(* PLC project Evolved Test, FAszom KFT TEST PLC Program 0.1.23.456 *)
(* stored: creationDateTime 1990-01-01T12:00:00, modificationDateTime 2016-04-10T17:37:00 *)

PROGRAM MotorExample
  VAR
    state : INT := 1;
    Distance : LREAL := 360;
    PowerX : MC_Power;
    Xonb : BOOL;
    HomeX : MC_Home;
    Referenced : BOOL;
    ExtendX : MC_MoveRelative;
    Wait : TON;
    RetractX : MC_MoveAbsolute;
    Wait_time : TIME := TIME#3s0ms;
    Elapsed_time : TIME;
    ResetX : MC_Reset;
    ReadAxisState : MC_ReadStatus;
    Xerrorstop : BOOL;
    XerrorID : DWORD;
    Counter : INT := 0;
  END_VAR
  VAR CONSTANT
    ERROR : INT := 99;
  END_VAR

                    
CASE state OF
	
1:
PowerX(
	Axis:=MotorExample_Motor , 
	Enable:=TRUE , 
	bRegulatorOn:=TRUE , 
	bDriveStart:=TRUE , 
	Status=> , 
	bRegulatorRealState=> , 
	bDriveStartRealState=> , 
	Busy=> , 
	Error=> , 
	ErrorID=> );
	
	IF PowerX.bDriveStartRealState THEN
		Xonb:=TRUE;
		state:=state+1;
		ELSE
			state:=ERROR;
	END_IF
	
2:
HomeX(
	Axis:=MotorExample_Motor , 
	Execute:=TRUE, 
	Position:=0.0, 
	Done=> , 
	Busy=> , 
	CommandAborted=> , 
	Error=> , 
	ErrorID=> );
		
	IF HomeX.Done THEN
		Referenced:=TRUE;
		state:=state+1;
		HomeX.Execute:=FALSE;
		ELSIF HomeX.Error OR Xerrorstop OR MotorExample_Motor.bError THEN
		state:=ERROR;
	END_IF
	
3:
ExtendX.Execute:=TRUE; 
ExtendX.Distance:=Distance; 
ExtendX.Velocity:=100; 
ExtendX.Acceleration:=1000; 
ExtendX.Deceleration:=1000; 
ExtendX.Jerk:=0; 

	IF ExtendX.Done THEN
		state:=state+1;
		ExtendX.Execute:=FALSE;
		ELSIF ExtendX.Error OR Xerrorstop OR MotorExample_Motor.bError THEN
		state:=ERROR;	
	END_IF
	
4:
Wait.IN:=TRUE;
Wait.PT:=Wait_time;
Elapsed_time:=Wait.ET;

	IF Wait.Q THEN
		state:=state+1;
		Wait.IN:=FALSE;
	END_IF

5: 
RetractX.Execute:=TRUE; 
RetractX.Position:=0; 
RetractX.Velocity:=100;
RetractX.Acceleration:=1000;
RetractX.Deceleration:=1000; 
RetractX.Jerk:=0; 

IF RetractX.Done THEN
		state:=state+1;
		RetractX.Execute:=FALSE;
		counter:=counter+1;
		ELSIF RetractX.Error OR Xerrorstop THEN
		state:=ERROR;
	END_IF
	
6: 
Wait.IN:=TRUE; 
Wait.PT:=Wait_time;
Elapsed_time:=Wait.ET;

	IF Wait.Q THEN
		state:=3;
		Wait.IN:=FALSE;
	END_IF
	
ERROR:
ResetX.Execute:=TRUE;
Wait.IN:=TRUE;
IF Wait.Q THEN
	ResetX.Execute:=FALSE;
	state:=1;
END_IF

END_CASE
ExtendX(Axis:=MotorExample_Motor);
Wait();
RetractX(Axis:=MotorExample_Motor);
ResetX(Axis:=MotorExample_Motor);
ReadAxisState(Axis:=MotorExample_Motor,Enable:=TRUE,ErrorStop=>Xerrorstop);




                  
END_PROGRAM

PROGRAM Motor_Proba
  VAR_INPUT
    START AT %MX0.1 : BOOL := FALSE;
    STOP AT %MX0.2 : BOOL := FALSE;
  END_VAR
  VAR
    MOTOR AT %MX1.0 : BOOL := FALSE;
    ERROR AT %MX2.0 : BOOL := FALSE;
  END_VAR
  VAR
    ERR_TIM : TON;
    EL_TIME : TIME;
  END_VAR
  VAR_OUTPUT
    ST_RED AT %QX1.1 : BOOL;
    ST_GREEN AT %QX3.1 : BOOL;
  END_VAR

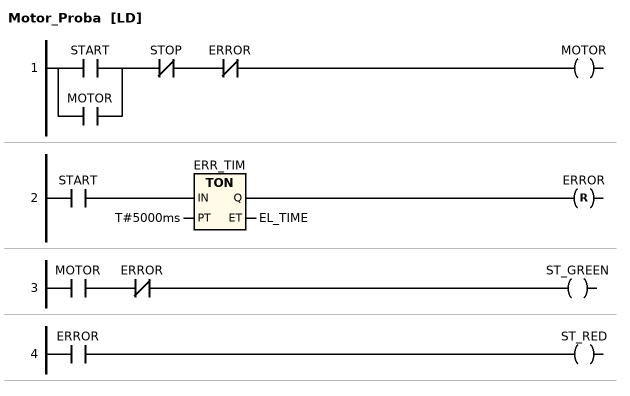
(* LD diagram, written out as Structured Text *)

MOTOR := (START OR MOTOR) AND NOT STOP AND NOT ERROR;

ERR_TIM(IN := START, PT := T#5000ms, ET => EL_TIME);
IF ERR_TIM.Q THEN ERROR := FALSE; END_IF;

ST_GREEN := MOTOR AND NOT ERROR;

ST_RED := ERROR;
END_PROGRAM

PROGRAM St_xample
  VAR
    input AT %MX3.3 : BOOL;
    output AT %QX0.1 : BOOL;
  END_VAR

									
									output := input;
									
								
END_PROGRAM

(* @NESTEDCOMMENTS := 'Yes' @PATH := '' @SYMFILEFLAGS := '2048' *)
FUNCTION_BLOCK fuzzy_exp
  VAR_INPUT
    PV : REAL;
    SP : REAL;
    MV_LN : REAL;
    MV_MN : REAL;
    MV_SN : REAL;
    MV_SP : REAL;
    MV_MP : REAL;
    MV_LP : REAL;
    LN_Error_Rate : REAL;
    MN_Error_Rate : REAL;
    MP_Error_Rate : REAL;
    LP_Error_Rate : REAL;
    Update_Time : WORD;
    Manual : BOOL;
    CV_Manual : REAL;
    CV_Min : REAL;
    CV_Max : REAL;
    Enable : BOOL;
  END_VAR
  VAR_OUTPUT
    FL_CV : REAL;
  END_VAR
  VAR
    Loop_Update_ONS : R_TRIG;
    Loop_Update_Trigger : BOOL;
    TMR_Loop_Update : TON;
    Loop_Update_Time : WORD;
    Loop_Update_mSec : TIME;
    Process_Error : REAL;
    NL_Error : BOOL;
    NM_Error : BOOL;
    NS_Error : BOOL;
    PS_Error : BOOL;
    PM_Error : BOOL;
    PL_Error : BOOL;
    Process_Error_Rate : REAL;
    Error_Rate_PV1 : REAL;
    Error_Rate_PV2 : REAL;
    NL_Error_Rate_Ind : BOOL;
    NM_Error_Rate_Ind : BOOL;
    NS_Error_Rate_Ind : BOOL;
    PS_Error_Rate_Ind : BOOL;
    PM_Error_Rate_Ind : BOOL;
    PL_Error_Rate_Ind : BOOL;
    Output_CV : REAL;
  END_VAR

                    (* @END_DECLARATION := '0' *)
(****************************************************************************************************************************
	POU Title:  	Fuzzy_Logic(PRG)
   
 	Designer:	K. Presssley
	Date:		01/09/09
		
	Function:	The function of this program is to implement a fuzzy logic control algorithm for process control..  
****************************************************************************************************************************)
(***** Loop Update Logic *****)
(*  Get the Loop Update Time, ensure that lower limit of 1 is not exceeded and convert it into a time variable  *)
	IF Update_Time < 1 THEN
		Loop_Update_Time := 1;
	ELSE
		Loop_Update_Time := Update_Time;
	END_IF;

	Loop_Update_mSec := WORD_TO_TIME(Loop_Update_Time);

	IF NOT TMR_Loop_Update.Q THEN
		Loop_Update_Trigger := TRUE;
	ELSE
		Loop_Update_Trigger := FALSE;
	END_IF;

	TMR_Loop_Update( IN := Loop_Update_Trigger, PT:= Loop_Update_mSec );
 	  Loop_Update_ONS( CLK := TMR_Loop_Update.Q);



(***** Calculate the Process Error and Process Error Rate *****)
	IF Loop_Update_ONS.Q THEN
	  (* Process Error Calculation *)
		Process_Error := SP - PV;

	  (* Process Error Rate Calculation *)
	 	Error_Rate_PV1 := Error_Rate_PV2;
		  Error_Rate_PV2 := PV;
		   Process_Error_Rate := (Error_Rate_PV2 - Error_Rate_PV1) / (Loop_Update_Time);
	END_IF;


(***** Membership Zone Logic *****)
(* Error Zone Identification Logic - This logic will indentify which Error Zone the Process Value is currently in *)
	(* Negative Large Membership Zone *)
		IF Process_Error <= MV_LN THEN
			NL_Error := TRUE;
		ELSE
			NL_Error := FALSE;
		END_IF;

	(* Negative Medium Membership Zone *)
		IF Process_Error > MV_LN AND Process_Error <= MV_MN THEN
			NM_Error := TRUE;
		ELSE
			NM_Error := FALSE;
		END_IF;

	(* Negative Small Membership Zone *)
		IF Process_Error > MV_MN AND Process_Error <= MV_SN THEN
			NS_Error := TRUE;
		ELSE
			NS_Error := FALSE;
		END_IF;

	(* Positive Small Membership Zone *)
		IF Process_Error < MV_MP AND Process_Error >= MV_SP THEN
			PS_Error := TRUE;
		ELSE
			PS_Error := FALSE;
		END_IF;

	(* Positive Medium Membership Zone *)
		IF Process_Error < MV_LP AND Process_Error >= MV_MP THEN
			PM_Error := TRUE;
		ELSE
			PM_Error := FALSE;
		END_IF;

	(* Positive Large Membership Zone *)
		IF Process_Error >= MV_LP THEN
			PL_Error := TRUE;
		ELSE
			PL_Error := FALSE;
		END_IF;

(* Error Rate Zone Identification Logic - This logic will indentify which Error Rate Zone the Process Value is currently in *)
	(* Negative Large Error Rate Membership Zone - The Error Rate is Decreasing Quickly *)
		IF Process_Error_Rate <= LN_Error_Rate THEN
			NL_Error_Rate_Ind := TRUE;
		ELSE
			NL_Error_Rate_Ind := FALSE;
		END_IF;

	(* Negative Medium Error Rate Membership Zone - The Error Rate is Decreasing *)
		IF Process_Error_Rate > LN_Error_Rate AND Process_Error_Rate <= MN_Error_Rate THEN
			NM_Error_Rate_Ind := TRUE;
		ELSE
			NM_Error_Rate_Ind := FALSE;
		END_IF;

	(* Negative Small Error Rate Membership Zone  - The Error Rate is Decreasing slowly *)
		IF Process_Error_Rate > MN_Error_Rate AND Process_Error_Rate < 0.0 THEN
			NS_Error_Rate_Ind := TRUE;
		ELSE
			NS_Error_Rate_Ind := FALSE;
		END_IF;

	(* Positive Small Error Rate Membership Zone  - The Error Rate is Increasing slowly *)
		IF Process_Error_Rate < MP_Error_Rate AND Process_Error_Rate >= 0.0 THEN
			PS_Error_Rate_Ind := TRUE;
		ELSE
			PS_Error_Rate_Ind := FALSE;
		END_IF;

	(* Positive Meduim Error Rate Membership Zone  - The Error Rate is Increasing *)
		IF Process_Error_Rate < LP_Error_Rate AND Process_Error_Rate >= MP_Error_Rate THEN
			PM_Error_Rate_Ind := TRUE;
		ELSE
			PM_Error_Rate_Ind := FALSE;
		END_IF;

	(* Positive Large Error Rate Membership Zone  - The Error Rate is Increasing Quickly  *)
		IF Process_Error_Rate >= LP_Error_Rate THEN
			PL_Error_Rate_Ind := TRUE;
		ELSE
			PL_Error_Rate_Ind := FALSE;
		END_IF;


(***** Fuzzy Logic Rules *****)
(* This section of logic contains all of the Fuzzy Logic rules required to produce the control action *)
	(* PV is Far Above SP and Increasing Quickly *)
		IF Loop_Update_ONS.Q AND NL_Error AND PL_Error_Rate_Ind
		    AND Enable AND NOT Manual THEN
			Output_CV := Output_CV - 1000.0;
		END_IF;

	(* PV is Far Above SP and Increasing *)
		IF Loop_Update_ONS.Q AND NL_Error AND PM_Error_Rate_Ind
		    AND Enable AND NOT Manual THEN
			Output_CV := Output_CV - 300.0;
		END_IF;

	(* PV is Far Above SP and Increasing slowly *)
		IF Loop_Update_ONS.Q AND NL_Error AND PS_Error_Rate_Ind
		    AND Enable AND NOT Manual THEN
			Output_CV := Output_CV - 250.0;
		END_IF;

	(* PV is Far Above SP and Decreasing slowly *)
		IF Loop_Update_ONS.Q AND NL_Error AND NS_Error_Rate_Ind
		    AND Enable AND NOT Manual THEN
			Output_CV := Output_CV - 300;
		END_IF;

	(* PV is Far Above SP and Decreasing *)
		IF Loop_Update_ONS.Q AND NL_Error AND NM_Error_Rate_Ind
		    AND Enable AND NOT Manual THEN
			Output_CV := Output_CV - 250.0;
		END_IF;

	(* PV is Far Above SP and Decreasing Quickly *)
		IF Loop_Update_ONS.Q AND NL_Error AND NL_Error_Rate_Ind
		    AND Enable AND NOT Manual THEN
			Output_CV := Output_CV - 100.0;
		END_IF;

	(* PV is Above SP and Increasing Quickly *)
		IF Loop_Update_ONS.Q AND NM_Error AND PL_Error_Rate_Ind
		    AND Enable AND NOT Manual THEN
			Output_CV := Output_CV - 250.0;
		END_IF;

	(* PV is Above SP and Increasing *)
		IF Loop_Update_ONS.Q AND NM_Error AND PM_Error_Rate_Ind
		    AND Enable AND NOT Manual THEN
			Output_CV := Output_CV - 100.0;
		END_IF;

	(* PV is Above SP and Increasing slowly *)
		IF Loop_Update_ONS.Q AND NM_Error AND PS_Error_Rate_Ind
		    AND Enable AND NOT Manual THEN
			Output_CV := Output_CV - 50.0;
		END_IF;

	(* PV is Above SP and Decreasing Slowly *)
		IF Loop_Update_ONS.Q AND NM_Error AND NS_Error_Rate_Ind
		    AND Enable AND NOT Manual THEN
			Output_CV := Output_CV - 250.0;
		END_IF;

	(* PV is Above SP and Decreasing *)
		IF Loop_Update_ONS.Q AND NM_Error AND NM_Error_Rate_Ind
		    AND Enable AND NOT Manual THEN
			Output_CV := Output_CV - 100.0;
		END_IF;

	(* PV is Above SP and Decreasing Quickly *)
		IF Loop_Update_ONS.Q AND NM_Error AND NL_Error_Rate_Ind
		    AND Enable AND NOT Manual THEN
			Output_CV := Output_CV - 50.0;
		END_IF;

	(* PV is Slightly Above SP and Increasing Quickly *)
		IF Loop_Update_ONS.Q AND NS_Error AND PL_Error_Rate_Ind
		    AND Enable AND NOT Manual THEN
			Output_CV := Output_CV - 20.0;
		END_IF;

	(* PV is Slightly Above SP and Increasing *)
		IF Loop_Update_ONS.Q AND NS_Error AND PM_Error_Rate_Ind
		    AND Enable AND NOT Manual THEN
			Output_CV := Output_CV - 10.0;
		END_IF;

	(* PV is Slightly Above SP and Increasing slowly*)
		IF Loop_Update_ONS.Q AND NS_Error AND PS_Error_Rate_Ind
		    AND Enable AND NOT Manual THEN
			Output_CV := Output_CV - 5.0;
		END_IF;

	(* PV is Slightly Above SP and Decreasing slowly*)
		IF Loop_Update_ONS.Q AND NS_Error AND NS_Error_Rate_Ind
		    AND Enable AND NOT Manual THEN
			Output_CV := Output_CV - 20.0;
		END_IF;

	(* PV is Slightly Above SP and Decreasing *)
		IF Loop_Update_ONS.Q AND NS_Error AND NM_Error_Rate_Ind
		    AND Enable AND NOT Manual THEN
			Output_CV := Output_CV - 10.0;
		END_IF;

	(* PV is Slightly Above SP and Decreasing Quickly*)
		IF Loop_Update_ONS.Q AND NS_Error AND NL_Error_Rate_Ind
		    AND Enable AND NOT Manual THEN
			Output_CV := Output_CV - 5.0;
		END_IF;

	(* PV is Slightly Below SP and Increasing Quickly *)
		IF Loop_Update_ONS.Q AND PS_Error AND PL_Error_Rate_Ind
		    AND Enable AND NOT Manual THEN
			Output_CV := Output_CV + 5.0;
		END_IF;

	(* PV is Slightly Below SP and Increasing *)
		IF Loop_Update_ONS.Q AND PS_Error AND PM_Error_Rate_Ind
		    AND Enable AND NOT Manual THEN
			Output_CV := Output_CV + 10.0;
		END_IF;

	(* PV is Slightly Below SP and Increasing Slowly *)
		IF Loop_Update_ONS.Q AND PS_Error AND PS_Error_Rate_Ind
		    AND Enable AND NOT Manual THEN
			Output_CV := Output_CV + 20.0;
		END_IF;

	(* PV is Slightly Below SP and Decreasing Slowly *)
		IF Loop_Update_ONS.Q AND PS_Error AND NS_Error_Rate_Ind
		    AND Enable AND NOT Manual THEN
			Output_CV := Output_CV + 20.0;
		END_IF;

	(* PV is Slightly Below SP and Decreasing *)
		IF Loop_Update_ONS.Q AND PS_Error AND NM_Error_Rate_Ind
		    AND Enable AND NOT Manual THEN
			Output_CV := Output_CV + 10.0;
		END_IF;

	(* PV is Slightly Below SP and Decreasing Quickly *)
		IF Loop_Update_ONS.Q AND PS_Error AND NL_Error_Rate_Ind
		    AND Enable AND NOT Manual THEN
			Output_CV := Output_CV + 5.0;
		END_IF;

	(* PV is Below SP and Increasing Quickly *)
		IF Loop_Update_ONS.Q AND PM_Error AND PL_Error_Rate_Ind
		    AND Enable AND NOT Manual THEN
			Output_CV := Output_CV + 50.0;
		END_IF;

	(* PV is Below SP and Increasing *)
		IF Loop_Update_ONS.Q AND PM_Error AND PM_Error_Rate_Ind
		    AND Enable AND NOT Manual THEN
			Output_CV := Output_CV + 20.0;
		END_IF;

	(* PV is Below SP and Increasing Slowly *)
		IF Loop_Update_ONS.Q AND PM_Error AND PS_Error_Rate_Ind
		    AND Enable AND NOT Manual THEN
			Output_CV := Output_CV + 10.0;
		END_IF;

	(* PV is Below SP and Decreasing Slowly *)
		IF Loop_Update_ONS.Q AND PM_Error AND NS_Error_Rate_Ind
		    AND Enable AND NOT Manual THEN
			Output_CV := Output_CV + 50.0;
		END_IF;

	(* PV is Below SP and Decreasing *)
		IF Loop_Update_ONS.Q AND PM_Error AND NM_Error_Rate_Ind
		    AND Enable AND NOT Manual THEN
			Output_CV := Output_CV + 100.0;
		END_IF;

	(* PV is Below SP and Decreasing Quickly *)
		IF Loop_Update_ONS.Q AND PM_Error AND NL_Error_Rate_Ind
		    AND Enable AND NOT Manual THEN
			Output_CV := Output_CV + 250.0;
		END_IF;

	(* PV is Far Below SP and Increasing Quickly *)
		IF Loop_Update_ONS.Q AND PL_Error AND PL_Error_Rate_Ind
		    AND Enable AND NOT Manual THEN
			Output_CV := Output_CV + 100.0;
		END_IF;

	(* PV is Far Below SP and Increasing *)
		IF Loop_Update_ONS.Q AND PL_Error AND PM_Error_Rate_Ind
		    AND Enable AND NOT Manual THEN
			Output_CV := Output_CV + 250.0;
		END_IF;

	(* PV is Far Below SP and Increasing Slowly *)
		IF Loop_Update_ONS.Q AND PL_Error AND PS_Error_Rate_Ind
		    AND Enable AND NOT Manual THEN
			Output_CV := Output_CV + 300.0;
		END_IF;

	(* PV is Far Below SP and Decreasing Slowly *)
		IF Loop_Update_ONS.Q AND PL_Error AND NS_Error_Rate_Ind
		    AND Enable AND NOT Manual THEN
			Output_CV := Output_CV + 100.0;
		END_IF;

	(* PV is Far Below SP and Decreasing *)
		IF Loop_Update_ONS.Q AND PL_Error AND NM_Error_Rate_Ind
		    AND Enable AND NOT Manual THEN
			Output_CV := Output_CV + 250.0;
		END_IF;

	(* PV is Far Below SP and Decreasing Quickly *)
		IF Loop_Update_ONS.Q AND PL_Error AND NL_Error_Rate_Ind
		    AND Enable AND NOT Manual THEN
			Output_CV := Output_CV + 300.0;
		END_IF;

	(* Write Output_CV to the controller output variable, CV *)
		IF Enable AND NOT Manual THEN
			FL_CV := Output_CV;
		END_IF;


(***** Fuzzy Logic Controller Maximum and Minimum Limits Logic *****)
(* Minimum Limits Logic *)
	IF Output_CV < CV_Min THEN
		Output_CV := CV_Min;
	END_IF;

(* Maximum Limits Logic *)
	IF Output_CV > CV_Max THEN
		Output_CV := CV_Max;
	END_IF;

(***** Manual Fuzzy Logic Controller Operation *****)
(* This section of logic controls the manual operation of the fuzzy logic controller.  If the controller
    is enabled and the manual control is set to True, then the output of the controller, CV, will be
    equal to CV_Manual. *)
	IF Enable AND Manual AND (CV_Manual > 0.0 AND CV_Manual <= 32767) THEN
		FL_CV := CV_Manual;
	END_IF;

	IF Enable AND Manual AND (CV_Manual < 0.0) THEN
		FL_CV := 0.0;
	END_IF;

	IF Enable AND Manual AND (CV_Manual >32767.0) THEN
		FL_CV := 32767.0;
	END_IF;

(* Fuzzy Logic Controller Enable Logic *)
	IF NOT Enable THEN
		Output_CV := 0.0;
		  FL_CV := 0.0;
	END_IF;

                  
END_FUNCTION_BLOCK

CONFIGURATION Evolved Test
  RESOURCE Application ON PLC
    TASK ExampleTask(INTERVAL := T#20ms, PRIORITY := 1);
    PROGRAM MotorExample WITH ExampleTask : MotorExample;
  END_RESOURCE
END_CONFIGURATION

CONFIGURATION EthernetModul11
END_CONFIGURATION
